// TwinCAT 3 PLC project Library02
// Title: MyLibrary02
// Company: MyCompany
// ProjectVersion: 1.0.0.0
// ProgramVersion: 3.1.4020.2
// libraries:
//   Tc2_Standard, * (Beckhoff Automation GmbH)
//   Tc2_System, * (Beckhoff Automation GmbH)
//   Tc3_Module, * (Beckhoff Automation GmbH)
// project tree:
//   / PlcTask.TcTTO
//   POUs/ FB_Foo.TcPOU
// (motion and I/O tree: see PLC project library01)
// real-time tasks:
//   TASK PlcTask: cycle T#10ms, priority 20, ADS port 350

CONFIGURATION Library02
    RESOURCE PLC ON TwinCAT3
        TASK PlcTask(INTERVAL := T#10ms, PRIORITY := 20);
    END_RESOURCE
END_CONFIGURATION

// ---- POUs/FB_Foo.TcPOU
FUNCTION_BLOCK PUBLIC FB_Foo
VAR_INPUT
END_VAR
VAR_OUTPUT
	{attribute 'init_namespace'}
	sNamespace	:	STRING;	
END_VAR
VAR
END_VAR

END_FUNCTION_BLOCK
